{attribute 'strict'}
TYPE E_CylinderError :
(
	CYLINDER_ERROR_OK						:= 0,	(*  *)
	CYLINDER_ERROR_MOVE_HOME_TIMED_OUT 		:= 10,	(*  *)
	CYLINDER_ERROR_MOVE_ACTIVE_TIMED_OUT 	:= 20	(*  *)
);
END_TYPE

(* stored: Version 1.1.0.1, ProductVersion 3.1.4024.12
   DUT E_CylinderError: Id {17434684-f67d-4dcb-abc4-c2fd105586c0} *)
